LIN {X 0,Y 31.217,Z 439.268,A -85,B 0,C 180,E1 -30413.525,E2 -30413.525} C_VEL
LIN {X 0,Y 30.664,Z 436.561,A -85,B 0,C 180,E1 -30418.347,E2 -30418.347} C_VEL
LIN {X 0,Y 30.593,Z 436.559,A -85,B 0,C 180,E1 -30421.839,E2 -30421.839} C_VEL
LIN {X 0,Y 30.094,Z 436.616,A -85,B 0,C 180,E1 -30433.493,E2 -30433.493} C_VEL
LIN {X 0,Y 29.859,Z 436.64,A -85,B 0,C 180,E1 -30439.553,E2 -30439.553} C_VEL
LIN {X 0,Y 29.492,Z 436.674,A -85,B 0,C 180,E1 -30448.45,E2 -30448.45} C_VEL
LIN {X 0,Y 29.546,Z 436.669,A -85,B 0,C 180,E1 -30465.51,E2 -30465.51} C_VEL
LIN {X 0,Y 29.524,Z 436.79,A -85,B 0,C 180,E1 -30483.089,E2 -30483.089} C_VEL
LIN {X 0,Y 30.301,Z 438.71,A -85,B 0,C 180,E1 -30488.057,E2 -30488.057} C_VEL
LIN {X 0,Y 32.985,Z 441.788,A -85,B 0,C 180,E1 -30497.652,E2 -30497.652} C_VEL
LIN {X 0,Y 34.893,Z 445.155,A -85,B 0,C 180,E1 -30504.183,E2 -30504.183} C_VEL
LIN {X 0,Y 36.54,Z 451.633,A -85,B 0,C 180,E1 -30512.228,E2 -30512.228} C_VEL
LIN {X 0,Y 37.799,Z 459.371,A -85,B 0,C 180,E1 -30520.675,E2 -30520.675} C_VEL
LIN {X 0,Y 38.345,Z 464.3,A -85,B 0,C 180,E1 -30525.869,E2 -30525.869} C_VEL
LIN {X 0,Y 37.709,Z 466.877,A -85,B 0,C 180,E1 -30528.177,E2 -30528.177} C_VEL
LIN {X 0,Y 32.751,Z 478.638,A -85,B 0,C 180,E1 -30540.89,E2 -30540.89} C_VEL
LIN {X 0,Y 29.43,Z 489.278,A -85,B 0,C 180,E1 -30558.967,E2 -30558.967} C_VEL
LIN {X 0,Y 28.84,Z 497.599,A -85,B 0,C 180,E1 -30578.58,E2 -30578.58} C_VEL
LIN {X 0,Y 31.783,Z 505.509,A -85,B 0,C 180,E1 -30600.011,E2 -30600.011} C_VEL
LIN {X 0,Y 38.19,Z 512.069,A -85,B 0,C 180,E1 -30616.134,E2 -30616.134} C_VEL
LIN {X 0,Y 47.765,Z 518.076,A -85,B 0,C 180,E1 -30628.085,E2 -30628.085} C_VEL
LIN {X 0,Y 48.68,Z 518.617,A -85,B 0,C 180,E1 -30630.041,E2 -30630.041} C_VEL
LIN {X 0,Y 38.884,Z 513.808,A -85,B 0,C 180,E1 -30643.757,E2 -30643.757} C_VEL
LIN {X 0,Y 32.994,Z 507.704,A -85,B 0,C 180,E1 -30664.836,E2 -30664.836} C_VEL
LIN {X 0,Y 32.386,Z 506.106,A -85,B 0,C 180,E1 -30670.409,E2 -30670.409} C_VEL
LIN {X 0,Y 31.64,Z 504.147,A -85,B 0,C 180,E1 -30676.244,E2 -30676.244} C_VEL
LIN {X 0,Y 29.859,Z 500.618,A -85,B 0,C 180,E1 -30684.336,E2 -30684.336} C_VEL
LIN {X 0,Y 27.787,Z 496.7,A -85,B 0,C 180,E1 -30692.249,E2 -30692.249} C_VEL
LIN {X 0,Y 25.503,Z 490.965,A -85,B 0,C 180,E1 -30704.058,E2 -30704.058} C_VEL
LIN {X 0,Y 25.221,Z 486.461,A -85,B 0,C 180,E1 -30713.614,E2 -30713.614} C_VEL
LIN {X 0,Y 25.552,Z 484.94,A -85,B 0,C 180,E1 -30716.709,E2 -30716.709} C_VEL
LIN {X 0,Y 26.549,Z 482.113,A -85,B 0,C 180,E1 -30722.031,E2 -30722.031} C_VEL
LIN {X 0,Y 27.195,Z 477.822,A -85,B 0,C 180,E1 -30729.149,E2 -30729.149} C_VEL
LIN {X 0,Y 28.988,Z 466.159,A -85,B 0,C 180,E1 -30744.998,E2 -30744.998} C_VEL
LIN {X 0,Y 31.051,Z 456.186,A -85,B 0,C 180,E1 -30754.977,E2 -30754.977} C_VEL
LIN {X 0,Y 28.96,Z 449.611,A -85,B 0,C 180,E1 -30766.304,E2 -30766.304} C_VEL
LIN {X 0,Y 28.01,Z 446.418,A -85,B 0,C 180,E1 -30772.773,E2 -30772.773} C_VEL
LIN {X 0,Y 26.954,Z 443.872,A -85,B 0,C 180,E1 -30779.987,E2 -30779.987} C_VEL
LIN {X 0,Y 25.786,Z 442.179,A -85,B 0,C 180,E1 -30787.818,E2 -30787.818} C_VEL
LIN {X 0,Y 24.72,Z 441.453,A -85,B 0,C 180,E1 -30796.502,E2 -30796.502} C_VEL
LIN {X 0,Y 23.995,Z 441.201,A -85,B 0,C 180,E1 -30808.391,E2 -30808.391} C_VEL
LIN {X 0,Y 23.945,Z 441.408,A -85,B 0,C 180,E1 -30815.926,E2 -30815.926} C_VEL
LIN {X 0,Y 25.465,Z 442.662,A -85,B 0,C 180,E1 -30836.429,E2 -30836.429} C_VEL
LIN {X 0,Y 28.781,Z 447.664,A -85,B 0,C 180,E1 -30855.814,E2 -30855.814} C_VEL
LIN {X 0,Y 29.823,Z 450.18,A -85,B 0,C 180,E1 -30861.366,E2 -30861.366} C_VEL
LIN {X 0,Y 30.714,Z 455.943,A -85,B 0,C 180,E1 -30869.952,E2 -30869.952} C_VEL
LIN {X 0,Y 31.381,Z 462.743,A -85,B 0,C 180,E1 -30879.109,E2 -30879.109} C_VEL
LIN {X 0,Y 31.493,Z 465.651,A -85,B 0,C 180,E1 -30882.846,E2 -30882.846} C_VEL
LIN {X 0,Y 26.361,Z 476.634,A -85,B 0,C 180,E1 -30895.901,E2 -30895.901} C_VEL
LIN {X 0,Y 22.652,Z 487.091,A -85,B 0,C 180,E1 -30917.005,E2 -30917.005} C_VEL
LIN {X 0,Y 22.176,Z 495.467,A -85,B 0,C 180,E1 -30941.725,E2 -30941.725} C_VEL
LIN {X 0,Y 26.126,Z 503.684,A -85,B 0,C 180,E1 -30967.744,E2 -30967.744} C_VEL
LIN {X 0,Y 33.75,Z 510.568,A -85,B 0,C 180,E1 -30984.624,E2 -30984.624} C_VEL
LIN {X 0,Y 38.067,Z 513.364,A -85,B 0,C 180,E1 -30990.081,E2 -30990.081} C_VEL
LIN {X 0,Y 28.51,Z 506.819,A -85,B 0,C 180,E1 -31012.023,E2 -31012.023} C_VEL
LIN {X 0,Y 25.849,Z 502.2,A -85,B 0,C 180,E1 -31030.193,E2 -31030.193} C_VEL
LIN {X 0,Y 25.025,Z 499.835,A -85,B 0,C 180,E1 -31037.902,E2 -31037.902} C_VEL
LIN {X 0,Y 24.096,Z 491.084,A -85,B 0,C 180,E1 -31062.698,E2 -31062.698} C_VEL
LIN {X 0,Y 25.552,Z 484.94,A -85,B 0,C 180,E1 -31076.709,E2 -31076.709} C_VEL
LIN {X 0,Y 26.017,Z 482.006,A -85,B 0,C 180,E1 -31082.266,E2 -31082.266} C_VEL
LIN {X 0,Y 25.884,Z 478.963,A -85,B 0,C 180,E1 -31087.656,E2 -31087.656} C_VEL
LIN {X 0,Y 24.738,Z 472.764,A -85,B 0,C 180,E1 -31098.686,E2 -31098.686} C_VEL
LIN {X 0,Y 23.798,Z 466.307,A -85,B 0,C 180,E1 -31110.534,E2 -31110.534} C_VEL
LIN {X 0,Y 24.199,Z 461.198,A -85,B 0,C 180,E1 -31118.572,E2 -31118.572} C_VEL
LIN {X 0,Y 24.633,Z 459.423,A -85,B 0,C 180,E1 -31120.747,E2 -31120.747} C_VEL
LIN {X 0,Y 24.759,Z 457.579,A -85,B 0,C 180,E1 -31123.495,E2 -31123.495} C_VEL
LIN {X 0,Y 23.665,Z 452.447,A -85,B 0,C 180,E1 -31135.727,E2 -31135.727} C_VEL
LIN {X 0,Y 23.053,Z 449.584,A -85,B 0,C 180,E1 -31144.36,E2 -31144.36} C_VEL
LIN {X 0,Y 22.644,Z 448.704,A -85,B 0,C 180,E1 -31148.92,E2 -31148.92} C_VEL
LIN {X 0,Y 21.742,Z 447.945,A -85,B 0,C 180,E1 -31158.841,E2 -31158.841} C_VEL
LIN {X 0,Y 21.278,Z 448.301,A -85,B 0,C 180,E1 -31181.323,E2 -31181.323} C_VEL
LIN {X 0,Y 21.711,Z 448.727,A -85,B 0,C 180,E1 -31189.564,E2 -31189.564} C_VEL
LIN {X 0,Y 22.391,Z 449.68,A -85,B 0,C 180,E1 -31197.86,E2 -31197.86} C_VEL
LIN {X 0,Y 24.269,Z 453.146,A -85,B 0,C 180,E1 -31213.104,E2 -31213.104} C_VEL
LIN {X 0,Y 24.681,Z 456.14,A -85,B 0,C 180,E1 -31219.549,E2 -31219.549} C_VEL
LIN {X 0,Y 24.939,Z 463.161,A -85,B 0,C 180,E1 -31231.959,E2 -31231.959} C_VEL
LIN {X 0,Y 24.768,Z 466.102,A -85,B 0,C 180,E1 -31236.677,E2 -31236.677} C_VEL
LIN {X 0,Y 19.439,Z 476.243,A -85,B 0,C 180,E1 -31251.113,E2 -31251.113} C_VEL
LIN {X 0,Y 15.663,Z 485.872,A -85,B 0,C 180,E1 -31277.728,E2 -31277.728} C_VEL
LIN {X 0,Y 16.287,Z 494.858,A -85,B 0,C 180,E1 -31314.78,E2 -31314.78} C_VEL
LIN {X 0,Y 23.026,Z 503.386,A -85,B 0,C 180,E1 -31343.863,E2 -31343.863} C_VEL
LIN {X 0,Y 27.122,Z 506.616,A -85,B 0,C 180,E1 -31351.23,E2 -31351.23} C_VEL
LIN {X 0,Y 25.91,Z 505.83,A -85,B 0,C 180,E1 -31355.637,E2 -31355.637} C_VEL
LIN {X 0,Y 20.442,Z 500.275,A -85,B 0,C 180,E1 -31379.042,E2 -31379.042} C_VEL
LIN {X 0,Y 19.185,Z 497.994,A -85,B 0,C 180,E1 -31388.594,E2 -31388.594} C_VEL
LIN {X 0,Y 17.206,Z 490.673,A -85,B 0,C 180,E1 -31415.947,E2 -31415.947} C_VEL
LIN {X 0,Y 19.316,Z 481.748,A -85,B 0,C 180,E1 -31443.167,E2 -31443.167} C_VEL
LIN {X 0,Y 20.132,Z 478.299,A -85,B 0,C 180,E1 -31450.982,E2 -31450.982} C_VEL
LIN {X 0,Y 22.361,Z 467.42,A -85,B 0,C 180,E1 -31470.598,E2 -31470.598} C_VEL
LIN {X 0,Y 24.633,Z 459.423,A -85,B 0,C 180,E1 -31480.747,E2 -31480.747} C_VEL
LIN {X 0,Y 24.606,Z 457.516,A -85,B 0,C 180,E1 -31484.029,E2 -31484.029} C_VEL
LIN {X 0,Y 23.533,Z 455.812,A -85,B 0,C 180,E1 -31489.713,E2 -31489.713} C_VEL
LIN {X 0,Y 22,Z 454.802,A -85,B 0,C 180,E1 -31496.69,E2 -31496.69} C_VEL
LIN {X 0,Y 19.935,Z 454.384,A -85,B 0,C 180,E1 -31507.648,E2 -31507.648} C_VEL
LIN {X 0,Y 18.045,Z 454.627,A -85,B 0,C 180,E1 -31536.359,E2 -31536.359} C_VEL
LIN {X 0,Y 18.46,Z 455.173,A -85,B 0,C 180,E1 -31549.559,E2 -31549.559} C_VEL
LIN {X 0,Y 19.189,Z 457.159,A -85,B 0,C 180,E1 -31563.16,E2 -31563.16} C_VEL
LIN {X 0,Y 19.419,Z 458.595,A -85,B 0,C 180,E1 -31568.702,E2 -31568.702} C_VEL
LIN {X 0,Y 18.812,Z 465.263,A -85,B 0,C 180,E1 -31584.332,E2 -31584.332} C_VEL
LIN {X 0,Y 18.554,Z 466.338,A -85,B 0,C 180,E1 -31586.332,E2 -31586.332} C_VEL
LIN {X 0,Y 11.852,Z 477.165,A -85,B 0,C 180,E1 -31605.625,E2 -31605.625} C_VEL
LIN {X 0,Y 8.502,Z 486.79,A -85,B 0,C 180,E1 -31654.957,E2 -31654.957} C_VEL
LIN {X 0,Y 11.687,Z 493.797,A -85,B 0,C 180,E1 -31697.53,E2 -31697.53} C_VEL
LIN {X 0,Y 17.434,Z 499.289,A -85,B 0,C 180,E1 -31716.414,E2 -31716.414} C_VEL
LIN {X 0,Y 14.281,Z 495.966,A -85,B 0,C 180,E1 -31732.168,E2 -31732.168} C_VEL
LIN {X 0,Y 10.567,Z 486.793,A -85,B 0,C 180,E1 -31779.713,E2 -31779.713} C_VEL
LIN {X 0,Y 12.976,Z 479.254,A -85,B 0,C 180,E1 -31812.765,E2 -31812.765} C_VEL
LIN {X 0,Y 15.917,Z 469.128,A -85,B 0,C 180,E1 -31839.615,E2 -31839.615} C_VEL
LIN {X 0,Y 19.037,Z 461.071,A -85,B 0,C 180,E1 -31852.024,E2 -31852.024} C_VEL
LIN {X 0,Y 19.199,Z 459.852,A -85,B 0,C 180,E1 -31854.73,E2 -31854.73} C_VEL
LIN {X 0,Y 19.091,Z 455.089,A -85,B 0,C 180,E1 -31870.598,E2 -31870.598} C_VEL
LIN {X 0,Y 18.346,Z 454.452,A -85,B 0,C 180,E1 -31882.503,E2 -31882.503} C_VEL
LIN {X 0,Y 18.045,Z 454.627,A -85,B 0,C 180,E1 -31896.359,E2 -31896.359} C_VEL
LIN {X 0,Y 17.855,Z 455.405,A -85,B 0,C 180,E1 -31902.173,E2 -31902.173} C_VEL
LIN {X 0,Y 17.057,Z 457.547,A -85,B 0,C 180,E1 -31907.822,E2 -31907.822} C_VEL
LIN {X 0,Y 14.34,Z 463.835,A -85,B 0,C 180,E1 -31919.445,E2 -31919.445} C_VEL
LIN {X 0,Y 13.748,Z 465.752,A -85,B 0,C 180,E1 -31925.262,E2 -31925.262} C_VEL
LIN {X 0,Y 13.139,Z 466.99,A -85,B 0,C 180,E1 -31927.304,E2 -31927.304} C_VEL
LIN {X 0,Y 4.816,Z 477.986,A -85,B 0,C 180,E1 -31942.159,E2 -31942.159} C_VEL
LIN {X 0,Y 3.654,Z 486.114,A -85,B 0,C 180,E1 -32072.432,E2 -32072.432} C_VEL
LIN {X 0,Y 5.051,Z 487.544,A -85,B 0,C 180,E1 -32081.799,E2 -32081.799} C_VEL
LIN {X 0,Y 4.332,Z 485.958,A -85,B 0,C 180,E1 -32109.33,E2 -32109.33} C_VEL
LIN {X 0,Y 6.264,Z 478.706,A -85,B 0,C 180,E1 -32187.729,E2 -32187.729} C_VEL
LIN {X 0,Y 11.057,Z 469.198,A -85,B 0,C 180,E1 -32222.03,E2 -32222.03} C_VEL
LIN {X 0,Y 14.318,Z 463.237,A -85,B 0,C 180,E1 -32230.436,E2 -32230.436} C_VEL
LIN {X 0,Y 14.758,Z 461.965,A -85,B 0,C 180,E1 -32234.004,E2 -32234.004} C_VEL
LIN {X 0,Y 15,Z 460.818,A -85,B 0,C 180,E1 -32240.154,E2 -32240.154} C_VEL
LIN {X 0,Y 14.581,Z 460.944,A -85,B 0,C 180,E1 -32253.07,E2 -32253.07} C_VEL
LIN {X 0,Y 14.795,Z 461.411,A -85,B 0,C 180,E1 -32267.457,E2 -32267.457} C_VEL
LIN {X 0,Y 14.704,Z 462.756,A -85,B 0,C 180,E1 -32276.185,E2 -32276.185} C_VEL
LIN {X 0,Y 14.34,Z 463.835,A -85,B 0,C 180,E1 -32279.445,E2 -32279.445} C_VEL
LIN {X 0,Y 14.17,Z 465.118,A -85,B 0,C 180,E1 -32281.191,E2 -32281.191} C_VEL
LIN {X 0,Y 14.17,Z 600,A -85,B 0,C 180,E1 -32281.191,E2 -32281.191} C_VEL
LIN {X 0,Y 14.17,Z 600,A -85,B 0,C 180,E1 -32281.191,E2 -32281.191}

QRS_NEXT_CUT()

QRS_NEXT()
QRS_HOME()

END
